            "DoorSideSidorAl-n" : Bool;   // ST2 Door sidoor Side - Output stage defective
            "DoorSideSidorAl-L" : Bool;   // ST2 Door sidoor Side - Current measurement error
            "DoorSideSidorAl-t" : Bool;   // ST2 Door sidoor Side - Belt torn
            "DoorSideSidorAl-U" : Bool;   // ST2 Door sidoor Side - Max. mass to be moved:
            "Spare 1_7" : Bool;
            CloseDoorByHand : Bool;   // ST2 Door sidoor Side - close by hand
            DoorFrontLearn : Bool;   // ST2 Doors side in learn procedure - Please Wait
            DoorSideSpecial : Bool;   // Please Wait - Sidoor Side in Special - mode The system is in an error state or special mode (system is shutting down, powering up or saving safety-related parameters)
            SidoorSideOpenAlarm : Bool;   // Sidoor Side - An obstruction was detected in the opening direction
            SidoorSideCloseAlarm : Bool;   // Sidoor Side - An obstruction was detected in the closing direction
            Temp1 : Array[4..9] of Byte;
         END_STRUCT;
         BASE : Struct   // SHUTTER
            ClampDownWP : Bool;   // ST2 Base Clamp down failed to advance I200.2/B274.8
            ClampDownPP : Bool;   // ST2 Base Clamp down failed to reverse I200.3/B274.10
            ClampDownBS : Bool;   // ST2 Base Clamp down both sensors ON I200.2-3/B274.8-10
            MobileBaseWP : Bool;   // ST2 Base Mobile base failed to advance I200.4/B274.12
            MobileBasePP : Bool;   // ST2 Base Mobile base failed to reverse I200.5/B274.14
            MobileBaseTS : Bool;   // ST2 Base Mobile base both sensors ON I200.4-5/B274.12-14
            ClampUpLeftWP : Bool;   // ST2 Base Clamp up left failed to advance I200.6/B274.16
            ClampUpLeftPP : Bool;   // ST2 Base Clamp up left failed to reverse I200.7/B274.18
            ClampUpLeftBS : Bool;   // ST2 Base Clamp up left both sensors ON I200.2-3/B274.16-18
            ClampUpRightWP : Bool;   // ST2 Base Clamp up right failed to advance I201.0/B275.4
            ClampUpRightPP : Bool;   // ST2 Base Clamp up right failed to reverse I201.1/B275.6
            ClampUpRightBS : Bool;   // ST2 Base Clamp up right both sensors ON I200.0-1/B275.4-6
            TankStopperWP : Bool;   // ST2 Tank Stopper failed to advance I231.4/B277.12
            TankStopperPP : Bool;   // ST2 Tank Stopper failed to reverse I231.5/B277.14
            TankStopperBS : Bool;   // ST2 Tank Stopper both sensors ON I231.4-5/B277.12-14
            Temp1 : Array[2..9] of Byte;
         END_STRUCT;
         ST2OP02 : Struct   // CUT FSU CONV
            UnitTransferAdvFlt : Bool;   // ST2OP02 (Cut FSU CONV) Unit Transfer Failed To Advance I220.0/B284.4
            UnitTransferRetFlt : Bool;   // ST2OP02 (Cut FSU CONV) Unit Transfer Failed To Return I220.1/B284.6
            UnitTransferTSFlt : Bool;   // ST2OP02 (Cut FSU CONV) Unit Transfer Two Sensors ON I220.0-1/B284.4-6
            CuttingAdvFlt : Bool;   // ST2OP02 (Cut FSU CONV) Cutting Cylinder Failed To Advance I220.2/B284.8
            CuttingRevFlt : Bool;   // ST2OP02 (Cut FSU CONV) Cutting Cylinder Failed To Return I220.3/B284.10
            CuttingTSFlt : Bool;   // ST2OP02 (Cut FSU CONV) Cutting Cylinder Two Sensors ON I220.2-3/B284.8-10
            ClampAdvFlt : Bool;   // ST2OP02 (Cut FSU CONV) Ring Clamp Failed To Advance I220.4/B284.12
            ClampRevFlt : Bool;   // ST2OP02 (Cut FSU CONV) Ring Clamp Failed To Return I220.5/B284.14
            ClampTSFlt : Bool;   // ST2OP02 (Cut FSU CONV) Ring Clamp Two Sensors ON I220.4-5/B284.12-14
            FingersAdvFlt : Bool;   // ST2OP02 (Cut FSU CONV) Fingers Failed To Advance I220.6/B284.16
            FingersRevFlt : Bool;   // ST2OP02 (Cut FSU CONV) Fingers Failed To Return I220.6/B284.16
            FingersTSFlt : Bool;
            Spare1_4Alm : Bool;
            Spare1_5Alm : Bool;
            Spare1_6Alm : Bool;
            Spare1_7Alm : Bool;
            SlugUnitFlt : Bool;   // ST2OP02 (Cut FSU CONV) Slug Not Detected on Unit RC300 I220.7/B284.18
            CuttingTimeOutFlt : Bool;   // ST2OP02 (Cut FSU CONV) Cutting Time Exceeded RC301
            CylFaultDuringCycleFlt : Bool;   // ST2OP02 (Cut FSU CONV) Cylinder Fault During Cycle RC302
            CycleNotFinishFlt : Bool;   // ST2OP02 (Cut FSU CONV) Cycle Failed To Finish RC303
            CycleNotStartedFlt : Bool;   // ST2OP02 (Cut FSU CONV) Cycle Not Started Fault RC304
            SlugFrameFlt : Bool;   // ST2OP02 (Cut FSU CONV) Slug Not Detected by Frame RC305 I201.3/B275.10
            CylPositionLostFlt : Bool;   // ST2OP02 (Cut FSU CONV) Cylinders Position Lost in manual RC306
            Spare2_7Alm : Bool;
            Spare3_0Alm : Bool;
            Spare3_1Alm : Bool;
            Spare3_2Alm : Bool;
            Spare3_3Alm : Bool;
            Spare3_4Alm : Bool;
            Spare3_5Alm : Bool;
            Spare3_6Alm : Bool;
            Spare3_7Alm : Bool;
            CircuitBreakerTripFlt : Bool;   // ST2OP02 (Cut FSU CONV) Circuit Breaker Tripped I26.0/F110.3
            SlugSensorOffFlt : Bool;   // ST2OP02 (Cut FSU CONV) Slug sensor OFF I220.7/B284.18
            ContactorOffFlt : Bool;   // ST2OP02 (Cut FSU CONV) Motor Contactor OFF I26.1/K145.3
            ContactorOnFlt : Bool;   // ST2OP02 (Cut FSU CONV) Motor Contactor ON I26.1/K145.3
            FrameConstantlyONFlt : Bool;   // ST2OP02 (Cut FSU CONV) Frame Constanly ON I201.3/B275.10
            ChangeKnife : Bool;   // ST2OP02 (Cut FSU CONV) Change knife
            Spare4_6Alm : Bool;
            Spare4_7Alm : Bool;
            CarStopWPAlm : Bool;   // ST2OP02 (Cut FSU CONV) Carriage stopper failed to advance I221.0/B285.4
            CarStopPPAlm : Bool;   // ST2OP02 (Cut FSU CONV) Carriage stopper failed to reverse I221.1/B285.6
            CarStopBSAlm : Bool;   // ST2OP02 (Cut FSU CONV) Carriage stopper both sensors ON I221.0-1/B285.4-6
            TrHorWPAlm : Bool;   // ST2OP02 (Cut FSU CONV) Tr horizontal failed to advance I221.2/B285.8
            TrHorPPAlm : Bool;   // ST2OP02 (Cut FSU CONV) Tr horizontal failed to reverse I221.3/B285.10
            TrHorBSAlm : Bool;   // ST2OP02 (Cut FSU CONV) Tr horizontal both sensors ON I221.2-3/B285.8-10
            Spare5_6Alm : Bool;
            SlugBoxFull : Bool;   // ST2OP02 (Cut FSU CONV) + ST2OP05 (CUT NIPPLE HV) Slug box full
            Temp1 : Array[6..9] of Byte;
         END_STRUCT;
         ST2OP03 : Struct   // NOTCHING
            TrHorAdvFlt : Bool;   // ST2OP03 (NOTCHING) Transfer Horizontal Failed To Advance I231.2/B277.8
            TrHorRetFlt : Bool;   // ST2OP03 (NOTCHING) Transfer Horizontal Failed To Return I231.3/B277.10
            TrHorTSFlt : Bool;   // ST2OP03 (NOTCHING) Transfer Horizontal Two Sensors ON I231.2-3/B277.8-10
            TrVerAdvFlt : Bool;   // ST2OP03 (NOTCHING) Transfer Vertical Failed To Advance I230.4/B276.12
            TrVerRetFlt : Bool;   // ST2OP03 (NOTCHING) Transfer Vertical Failed To Return I230.5/B276.14
            TrVerTSFlt : Bool;   // ST2OP03 (NOTCHING) Transfer Vertical Two Sensors ON I230.4-5/B276.12-14
            RotAdvFlt : Bool;   // ST2OP03 (NOTCHING) Rotation Failed To Advance I230.2/B276.8
            RotRetFlt : Bool;   // ST2OP03 (NOTCHING) Rotation Failed To Return I230.3/B276.10
            RotTSFlt : Bool;   // ST2OP03 (NOTCHING) Rotation Two Sensors ON I230.2-3/B276.8-10
            StampArmAdvFlt : Bool;   // ST2OP03 (NOTCHING) Stamp Arm Failed To Advance I231.6/B277.16
            StampArmRetFlt : Bool;   // ST2OP03 (NOTCHING) Stamp Arm Failed To Return I231.7/B277.18
            StampArmTSFlt : Bool;   // ST2OP03 (NOTCHING) Stamp Arm Two Sensors ON I231.6-8/B277.16-18
            StampAdvFlt : Bool;   // ST2OP03 (NOTCHING) Cutting Cylinder Failed To Advance I230.0/B276.4
            StampRevFlt : Bool;   // ST2OP03 (NOTCHING) Cutting Cylinder Failed To Return I230.1/B276.6
            StampTSFlt : Bool;   // ST2OP03 (NOTCHING) Cutting Cylinder Two Sensors ON I230.0-1/B276.4-6
            OperationNotCompletedCorrectlyFlt : Bool;   // ST2OP03 (NOTCHING) Operation not completed correctly RC1601
            Slug1DetectionFlt : Bool;   // ST2OP03 (NOTCHING) Slug 1 Detection on Unit Fault I230.6/B276.16 RC1600
            Slug2DetectionFlt : Bool;   // ST2OP03 (NOTCHING) Slug 2 Detection on Unit Fault I230.7/B276.18 RC1600
            Slug1StillPresent : Bool;   // ST2OP03 (NOTCHING) Slug 1 stuck in blowing system
            Slug2StillPresent : Bool;   // ST2OP03 (NOTCHING) Slug 2 stuck in blowing system
            CycleNotStarted : Bool;   // ST2OP03 (NOTCHING) Cycle Not Started
            CycleNotFinished : Bool;   // ST2OP03 (NOTCHING) Cycle Not Finished
            CycleTime : Bool;   // ST2OP03 (NOTCHING) Cycle Time too long
            Presence : Bool;   // ST2OP03 (NOTCHING) Alarm Presence
            Temp1 : Array[6..11] of Byte;
         END_STRUCT;
         ST2OP04 : Struct   // WELD / WELD FB CONV
            HeaterTransferAdvFlt : Bool;   // ST2OP04 (WELD FB CONV) Heater Transfer Failed to Advance I240.6/B293.16
            HeaterTransferRetFlt : Bool;   // ST2OP04 (WELD FB CONV) Heater Transfer Failed to Return I240.7/B293.18
            HeaterTransferTSFlt : Bool;   // ST2OP04 (WELD FB CONV) Heater Transfer Two Sensors on I240.6-7/B293.16-18
            GcylAdvHeatingFlt : Bool;   // ST2OP04 (WELD FB CONV) Gcyl Failed to Advance Heating I240.2/B293.8
            GcylAdvCoolingFlt : Bool;   // ST2OP04 (WELD FB CONV) Gcyl Failed to Advance Cooling I240.1/B293.6
            GcylAdvLoadingFlt : Bool;   // ST2OP04 (WELD FB CONV) Gcyl Failed to Advance Loading I240.0/B293.4
            GcylRetFlt : Bool;   // ST2OP04 (WELD FB CONV) Gcyl Failed to Return I240.3/B293.10
            GcylTSFlt : Bool;   // ST2OP04 (WELD FB CONV) Gcyl Two Sensors on I240.0/B293.4-I240.3/B293.10
            HcylAdvFlt : Bool;   // ST2OP04 (WELD FB CONV) Hcyl Failed to Advance I240.4/B293.12 (Ret Sensor for BC)
            HcylRevFlt : Bool;   // ST2OP04 (WELD FB CONV) Hcyl Failed to Return I240.5/B293.14
            HcylTSFlt : Bool;   // ST2OP04 (WELD FB CONV) Hcyl Two Sensors on I240.4/B293.12- I240.5/B293.14
            GripperAdvGripFlt : Bool;   // ST2OP04 (WELD FB CONV) Gripper Failed to Grip (Ungrip sensor Fault) I240.1/B257.4
            GripperRetUngripFlt : Bool;   // ST2OP04 (WELD FB CONV) Gripper Failed to Ungrip Sensor Fault I240.1/B257.4
            GripTSFlt : Bool;   // not used
            SpareCylFaultsInt0 : Int;
            SpareCylFaultsDInt0 : DInt;
            CompHeatPosFlt : Bool;   // ST2OP04 (WELD FB CONV) Component Failed To Gcyl Heating Position I240.2/B293.8 RC201/101
            TankHeatPosFlt : Bool;   // ST2OP04 (WELD FB CONV) Hotplate Failed To Hcyl Heating Position I240.4/B293.12 RC217
            CompCoolPosFlt : Bool;   // ST2OP04 (WELD FB CONV) Component Failed To Gcyl Cooling Position I240.1/B293.6 RC202/102
            OpenTimeFlt : Bool;   // ST2OP04 (WELD FB CONV) Open Time Exceeded RC203/103
            TempDuringCycleFlt : Bool;   // ST2OP04 (WELD FB CONV) Hotplate Temperature Fault During Cycle RC204/104
            ReservedRC0_5 : Bool;
            CompHeatPressFlt : Bool;   // ST2OP04 (WELD FB CONV) Component Heating Pressure Out Of Tolerance RC205/105
            ReservedRC0_7 : Bool;
            CompCoolPressFlt : Bool;   // ST2OP04 (WELD FB CONV) Component Cooling Pressure Out Of Tolerance RC206/106
            ReservedRC1_1 : Bool;
            ReservedRC1_2 : Bool;
            ReservedRC1_3 : Bool;
            ReservedRC1_4 : Bool;
            ReservedRC1_5 : Bool;
            TankHeatPressFlt : Bool;   // ST2OP04 (WELD FB CONV) Hcyl Heating Pressure Out Of Tolerance RC207/107
            ReservedRC1_7 : Bool;
            ReservedRC2_0 : Bool;
            ReservedRC2_1 : Bool;
            ReservedRC2_2 : Bool;
            ReservedRC2_3 : Bool;
            CycleNotFinishFlt : Bool;   // ST2OP04 (WELD FB CONV) Cycle Failed To Finish RC211/111
            CycleNotStartedFlt : Bool;   // ST2OP04 (WELD FB CONV) Cycle Not Started Fault RC212/112
            ReservedRC2_6 : Bool;
            ReservedRC2_7 : Bool;
            ReservedRC3_0 : Bool;
            TankHeatContactFlt : Bool;   // ST2OP04 (WELD FB CONV) Tank Heating Contact Pressure Calc Out Of Tolerance RC213/113
            ReservedRC3_2 : Bool;
            ReservedRC3_3 : Bool;
            MeltedComponentFlt : Bool;   // ST2OP04 (WELD FB CONV) Remove Melted Component From Gripper I241.2/B294.8 RC214/114
            ReservedRC3_5 : Bool;
            CylFaultDuringCycleFlt : Bool;   // ST2OP04 (WELD FB CONV) Cylinder Fault During Cycle RC215/115
            ReservedRC3_7 : Bool;
            ManualUsedFlt : Bool;   // ST2OP04 (WELD FB CONV) Manual Movements Used RC216/116
            CompPresent1AfterHeatFlt : Bool;   // ST2OP04 (WELD FB CONV) Component Present 1 Missing After Heating I241.2/B294.8 RC208/108
            CompPresent2AfterHeatFlt : Bool;   // ST2OP04 (WELD FB CONV) Component Present 2 Missing After Heating XXX RC218/118
            CompPresent3AfterHeatFlt : Bool;   // ST2OP04 (WELD FB CONV) Component Present 3 Missing After Heating Ixx.X RC219/119
            CompPresent4AfterHeatFlt : Bool;   // ST2OP04 (WELD FB CONV) Component Present 4 Missing After Heating Ixx.X RC220/240
            CompPresent5AfterHeatFlt : Bool;   // ST2OP04 (WELD FB CONV) Component Present 5 Missing After Heating Ixx.X RC221/121
            CompPresent6AfterHeatFlt : Bool;   // ST2OP04 (WELD FB CONV) Component Present 6 Missing After Heating Ixx.X RC222/122
            CompPresent7AfterHeatFlt : Bool;   // ST2OP04 (WELD FB CONV) Component Present 7 Missing After Heating Ixx.X RC223/123
            CompPresent8AfterHeatFlt : Bool;   // ST2OP04 (WELD FB CONV) Component Present 8 Missing After Heating Ixx.X RC224/124
            RemoveComponent1Flt : Bool;   // ST2OP04 (WELD FB CONV) Remove Component From Gripper (Present 1 after welding) I241.2/B294.8 RC209/109
            RemoveComponent2Flt : Bool;   // ST2OP04 (WELD FB CONV) Remove Component From Gripper (Present 2 after welding) XXX RC225/125
            RemoveComponent3Flt : Bool;   // ST2OP04 (WELD FB CONV) Remove Component From Gripper (Present 3 after welding) Ixx.X RC226/126
            RemoveComponent4Flt : Bool;   // ST2OP04 (WELD FB CONV) Remove Component From Gripper (Present 4 after welding) Ixx.X RC227/127
            RemoveComponent5Flt : Bool;   // ST2OP04 (WELD FB CONV) Remove Component From Gripper (Present 5 after welding) Ixx.X RC228/128
            RemoveComponent6Flt : Bool;   // ST2OP04 (WELD FB CONV) Remove Component From Gripper (Present 6 after welding) Ixx.X RC229/129
            RemoveComponent7Flt : Bool;   // ST2OP04 (WELD FB CONV) Remove Component From Gripper (Present 7 after welding) Ixx.X RC230/130
            RemoveComponent8Flt : Bool;   // ST2OP04 (WELD FB CONV) Remove Component From Gripper (Present 8 after welding) Ixx.X RC231/131
            CompMissing1Flt : Bool;   // ST2OP04 (WELD FB CONV) Component Present 1 Missing In Gripper I241.2/B294.8 RC210/110
            CompMissing2Flt : Bool;   // ST2OP04 (WELD FB CONV) Component Present 2 Missing In Gripper XXX RC232/132
            CompMissing3Flt : Bool;   // ST2OP04 (WELD FB CONV) Component Present 3 Missing In Gripper Ixx.X RC233/133
            CompMissing4Flt : Bool;   // ST2OP04 (WELD FB CONV) Component Present 4 Missing In Gripper Ixx.X RC234/134
            CompMissing5Flt : Bool;   // ST2OP04 (WELD FB CONV) Component Present 5 Missing In Gripper Ixx.X RC235/135
            CompMissing6Flt : Bool;   // ST2OP04 (WELD FB CONV) Component Present 6 Missing In Gripper Ixx.X RC236/136
            CompMissing7Flt : Bool;   // ST2OP04 (WELD FB CONV) Component Present 7 Missing In Gripper Ixx.X RC237/137
            CompMissing8Flt : Bool;   // ST2OP04 (WELD FB CONV) Component Present 8 Missing In Gripper Ixx.X RC238/138
            SpareFaultRC : Byte;
            HotplateTempOutFlt : Bool;   // ST2OP04 (WELD FB CONV) Hotplate Temperature Out Of Tolerance
            HotplateTempSensorFlt : Bool;   // ST2OP04 (WELD FB CONV) Hotplate Thermocouple Wire Break
            HotplateTempDiffereneceTooBigFlt : Bool;   // ST2OP04 (WELD FB CONV) Hotplate Thermocouples Difference Too Big
            Reserved0_3 : Bool;
            Reserved0_4 : Bool;
            Reserved0_5 : Bool;
            CompStuckOnTankFlt : Bool;   // ST2OP04 (WELD FB CONV) Component Stuck On Tank Must reset to Ungrip Component
            TempSetFlt : Bool;   // ST2OP04 (WELD FB CONV) Hotplate Tempearture Setpoint Out Of Range
            Reserved1_0 : Bool;
            RemoveHeatedComponentFlt : Bool;   // ST2OP04 (WELD FB CONV) Remove Heated Component
            CleanHotplatesFlt : Bool;   // ST2OP04 (WELD FB CONV) Clean Hotplates
            NoDetectionUsed : Bool;   // ST2OP04 (WELD FB CONV) No Detection Used (PLC program issue)
            SpareAlarmsDInt0 : DInt;
            HotTempChanFlt : Bool;   // ST2OP04 (WELD FB CONV) Hotplate Temperature is not changing
            Spare_1 : Bool;
            Spare_2 : Bool;
            Spare_3 : Bool;
            Spare_4 : Bool;
            Spare_5 : Bool;
            Spare_6 : Bool;
            Spare_7 : Bool;
            Spare_8 : Bool;
            Spare_9 : Bool;
            Spare_10 : Bool;
            Spare_11 : Bool;
            Spare_12 : Bool;
            Spare_13 : Bool;
            Spare_14 : Bool;
            Spare_15 : Bool;
            TrCrossdvFlt : Bool;   // ST2OP04 (WELD FB CONV) Transfer Cross failed to advance I241.4/B294.12
            TrCrossRevFlt : Bool;   // ST2OP04 (WELD FB CONV) Transfer Cross failed to reverse I241.5/B294.14
            TrCrossTsFlt : Bool;   // ST2OP04 (WELD FB CONV) Transfer Cross both sensors ON I241.4-5-2/B294.12-14
            Spare_19 : Bool;
            Spare_21 : Bool;
            Spare_20 : Bool;
            TrCrossdvFlt_1 : Bool;   // ST2OP04 (WELD FB CONV) Stopper Tr Cross failed to advance I241.6/B294.16
            TrCrossRevFlt_1 : Bool;   // ST2OP04 (WELD FB CONV) Stopper Tr Cross failed to reverse I241.7/B294.18
            TrCrossTsFlt_1 : Bool;   // ST2OP04 (WELD FB CONV) Stopper Tr Cross both sensors ON I241.6-7/B294.16-18
            Spare_25 : Bool;
            Spare_26 : Bool;
            Spare_27 : Bool;
            Spare_28 : Bool;
            Spare_29 : Bool;
            Spare_30 : Bool;
            Spare_31 : Bool;
            RemCycleNotStartedBADFromPrevStation : Bool;
            Spare_33 : Bool;
            Spare_34 : Bool;
            FailedToAutoLoad : Bool;
            Spare_36 : Bool;
            Spare_37 : Bool;
            Spare_38 : Bool;
         END_STRUCT;
         ST2OP05 : Struct   // CUT NIPPLE HV
            UnitTransferAdvFlt : Bool;   // ST2OP05 (CUT NIPPLE HV) Unit Transfer Failed To Advance I250.0/B286.4
            UnitTransferRetFlt : Bool;   // ST2OP05 (CUT NIPPLE HV) Unit Transfer Failed To Return I250.1/B286.6
            UnitTransferTSFlt : Bool;   // ST2OP05 (CUT NIPPLE HV) Unit Transfer Two Sensors ON I250.0-1/B286.4-6
            CuttingAdvFlt : Bool;   // ST2OP05 (CUT NIPPLE HV) Cutting Cylinder Failed To Advance I250.2/B286.8
            CuttingRevFlt : Bool;   // ST2OP05 (CUT NIPPLE HV) Cutting Cylinder Failed To Return I250.3/B286.10
            CuttingTSFlt : Bool;   // ST2OP05 (CUT NIPPLE HV) Cutting Cylinder Two Sensors ON I250.2-3/B286.8-10
            NeedleAdvFlt : Bool;   // ST2OP05 (CUT NIPPLE HV) Slug Needle Failed To Advance I250.4/B286.12
            NeedleRevFlt : Bool;   // ST2OP05 (CUT NIPPLE HV) Slug Needle Failed To Return I250.5/B286.14
            NeedleTSFlt : Bool;   // ST2OP05 (CUT NIPPLE HV) Slug Needle Two Sensors ON I250.4-5/B286.12-14
            SpareCylFaults : Int;
            SlugUnitFlt : Bool;   // ST2OP05 (CUT NIPPLE HV) Slug Not Detected on Unit RC350 I250.6/B286.16
            CuttingTimeOutFlt : Bool;   // ST2OP05 (CUT NIPPLE HV) Cutting Time Exceeded RC351
            CylFaultDuringCycleFlt : Bool;   // ST2OP05 (CUT NIPPLE HV) Cylinder Fault During Cycle RC352
            CycleNotFinishFlt : Bool;   // ST2OP05 (CUT NIPPLE HV) Cycle Failed To Finish RC353
            CycleNotStartedFlt : Bool;   // ST2OP05 (CUT NIPPLE HV) Cycle Not Started Fault RC354
            SlugFrameFlt : Bool;   // ST2OP05 (CUT NIPPLE HV) Slug Not Detected by Frame RC355 I201.3/B275.10
            ManualUsedFlt : Bool;   // ST2OP05 (CUT NIPPLE HV) Cylinders Position Lost in manual RC356
            Spare2_7Alm : Bool;
            Spare3_0Alm : Bool;
            BumperHorizontalWPAlm : Bool;
            BumperHorizontalPPAlm : Bool;
            BumperHorizontalBSAlm : Bool;
            Spare_8_7Alm : Bool;
            MissingStartFromSTDBlock : Bool;   // ST2OP05 (CUT NIPPLE HV) Missing Start Cycle From Standard Block
            SlugBoxFull : Bool;
            Spare3_7Alm : Bool;
            CircuitBreakerTripFlt : Bool;   // ST2OP05 (CUT NIPPLE HV) Circuit Breaker Tripped I26.2/F110.7
            SlugSensorOnFlt : Bool;   // ST2OP05 (CUT NIPPLE HV) Slug sensor ON I250.6/B286.16
            ContactorOffFlt : Bool;   // ST2OP05 (CUT NIPPLE HV) Motor Contactor OFF I26.3/K145.5
            ContactorOnFlt : Bool;   // ST2OP05 (CUT NIPPLE HV) Motor Contactor ON I26.3/K145.5
            FrameConstantlyONFlt : Bool;   // ST2OP05 (CUT NIPPLE HV) Frame Constanly ON I201.3/B275.10
            ChangeKnife : Bool;   // ST2OP05 (CUT NIPPLE HV) Change knife
            Spare4_6Alm : Bool;
            Spare4_7Alm : Bool;
            CarStopWPAlm : Bool;   // ST2OP05 (CUT NIPPLE HV) Carriage stopper failed to advance I251.0/B287.4
            CarStopPPAlm : Bool;   // ST2OP05 (CUT NIPPLE HV) Carriage stopper failed to reverse I251.1/B287.6
            CarStopBSAlm : Bool;   // ST2OP05 (CUT NIPPLE HV) Carriage stopper both sensors on I251.0-1/B287.4-6
            HorizontalTrAdvFlt : Bool;   // ST2OP05 (CUT NIPPLE HV) Transfer Horizontal failed to advance I251.2/B287.8
            HorizontalTrRetFlt : Bool;   // ST2OP05 (CUT NIPPLE HV) Transfer Horizontal failed to reverse I251.3/B287.10
            HorizontalTrTSFlt : Bool;   // ST2OP05 (CUT NIPPLE HV) Transfer Horizontal both sensors ON I251.2-3 /B287.8-10
            Spare7_6Alm : Bool;
            Spare7_7Alm : Bool;
            Spare8_0Alm : Bool;
            VacuumFlapWP : Bool;
            VacuumFlapPP : Bool;
            VacuumFlapBS : Bool;
            Spare7_6Alm_2 : Bool;
            Spare7_7Alm_2 : Bool;
            Spare8_0Alm_2 : Bool;
            Spare7_6Alm_3 : Bool;
            Spare7_7Alm_3 : Bool;
            Spare8_0Alm_3 : Bool;
            Spare7_6Alm_4 : Bool;
            Spare7_7Alm_4 : Bool;
            Spare8_0Alm_4 : Bool;
            Spare8_0Alm_5 : Bool;
            Spare8_0Alm_6 : Bool;
            Spare8_0Alm_7 : Bool;
         END_STRUCT;
         ST2OP06 : Struct   // WELD ICV HV
            HeaterTransferAdvFlt : Bool;   // ST2OP06 (WELD ICV HV) Heater Transfer Failed to Advance I260.6/B295.16
            HeaterTransferRetFlt : Bool;   // ST2OP06 (WELD ICV HV) Heater Transfer Failed to Return I260.7/B295.18
            HeaterTransferTSFlt : Bool;   // ST2OP06 (WELD ICV HV) Heater Transfer Two Sensors on I260.6-7/B295.16-18
            GcylAdvHeatingFlt : Bool;   // ST2OP06 (WELD ICV HV) Gcyl Failed to Advance Heating I260.2/B295.8
            GcylAdvCoolingFlt : Bool;   // ST2OP06 (WELD ICV HV) Gcyl Failed to Advance Cooling I260.1/B295.6
            GcylAdvLoadingFlt : Bool;   // ST2OP06 (WELD ICV HV) Gcyl Failed to Advance Loading I260.0/B295.4
            GcylRetFlt : Bool;   // ST2OP06 (WELD ICV HV) Gcyl Failed to Return I260.3/B295.10
            GcylTSFlt : Bool;   // ST2OP06 (WELD ICV HV) Gcyl Two Sensors on I260.0-3/B295.4-10
            HcylAdvFlt : Bool;   // ST2OP06 (WELD ICV HV) Hcyl Failed to Advance I260.4/B295.12
            HcylRevFlt : Bool;   // ST2OP06 (WELD ICV HV) Hcyl Failed to Return I260.5/B295.14
            HcylTSFlt : Bool;   // ST2OP06 (WELD ICV HV) Hcyl Two Sensors on I260.4-5/B295.12-14
            GripperAdvGripFlt : Bool;   // ST2OP06 (WELD ICV HV) Gripper Failed to Grip (Ungrip sensor Fault) I261.0/B296.4
            GripperRetUngripFlt : Bool;   // ST2OP06 (WELD ICV HV) Gripper Failed to Ungrip Sensor Fault I261.0/B296.4
            GripTSFlt : Bool;   // not used
            ApproachGcylAdvFlt : Bool;   // ST2OP06 (WELD ICV HV) Approach Gcyl Failed to Advance Ix.x
            ApproachGcylRetFlt : Bool;   // ST2OP06 (WELD ICV HV) Approach Gcyl Failed to Return Ix.x
            ApproachGcylTSFlt : Bool;   // ST2OP06 (WELD ICV HV) Approach Gcyl Two Sensors on Ixx.X-Ixx.X
            ApproachHcylAdvFlt : Bool;   // ST2OP06 (WELD ICV HV) Approach Hcyl Failed to Advance Ix.x
            ApproachHcylRetFlt : Bool;   // ST2OP06 (WELD ICV HV) Approach Hcyl Failed to Return Ix.x
            ApproachHcylTSFlt : Bool;   // ST2OP06 (WELD ICV HV) Approach Hcyl Two Sensors on Ixx.X-Ixx.X
            ComplGcylAdvLockFlt : Bool;   // ST2OP06 (WELD ICV HV) Compliancy Gcyl Failed to Lock Ix.x
            ComplGcylRetUnlockFlt : Bool;   // ST2OP06 (WELD ICV HV) Compliancy Gcyl Failed to Unlock Ix.x
            ComplGcylRetTSFlt : Bool;   // ST2OP06 (WELD ICV HV) Compliancy Gcyl Two Sensors on Ixx.X-Ixx.X
            ComplHcylAdvLockFlt : Bool;   // ST2OP06 (WELD ICV HV) Compliancy Hcyl Failed to Lock Ix.x
            ComplHcylRetUnlockFlt : Bool;   // ST2OP06 (WELD ICV HV) Compliancy Hcyl Failed to Unlock Ix.x
            ComplHcylRetTSFlt : Bool;   // ST2OP06 (WELD ICV HV) Compliancy Hcyl Two Sensors on Ixx.X-Ixx.X
            ComponentHeaterAdvFlt : Bool;   // ST2OP06 (WELD ICV HV) Component Heater Failed to Advance Ixx.X
            ComponentHeaterRetFlt : Bool;   // ST2OP06 (WELD ICV HV) Component Heater Failed to Return Ixx.X
            ComponentHeaterTSFlt : Bool;   // ST2OP06 (WELD ICV HV) Component Heater Two Sensors on Ixx.X-Ixx.X
            PullerAdvFlt : Bool;   // ST2OP06 (WELD ICV HV) Puller Failed to Advance Ixx.X
            PullerRetFlt : Bool;   // ST2OP06 (WELD ICV HV) Puller Failed to Return Ixx.X
            PullerTSFlt : Bool;   // ST2OP06 (WELD ICV HV) Puller Two Sensors on Ixx.X-Ixx.X
            SpareCylFaultsDInt0 : DInt;
            CompHeatPosFlt : Bool;   // ST2OP06 (WELD ICV HV) Component Failed To Gcyl Heating Position I260.2/B295.8 RC001
            TankHeatPosFlt : Bool;   // ST2OP06 (WELD ICV HV) Tank Hotplate Failed To Hcyl Heating Position I260.4/B295.12 RC002
            CompCoolPosFlt : Bool;   // ST2OP06 (WELD ICV HV) Component Failed To Gcyl Cooling Position I260.1/B295.6 RC003
            OpenTimeFlt : Bool;   // ST2OP06 (WELD ICV HV) Open Time Exceeded RC004
            TankTempDuringCycleFlt : Bool;   // ST2OP06 (WELD ICV HV) Tank Hotplate Temperature Fault During Cycle RC005
            CompMatchForwPressFlt : Bool;   // ST2OP06 (WELD ICV HV) Component Matching Forward Pressure Out Of Tolerance RC006
            CompHeatForwPressFlt : Bool;   // ST2OP06 (WELD ICV HV) Component Heating Forward Pressure Out Of Tolerance RC007
            CompJunctForwPressFlt : Bool;   // ST2OP06 (WELD ICV HV) Component Junction Forward Pressure Out Of Tolerance RC008
            CompCoolForwPressFlt : Bool;   // ST2OP06 (WELD ICV HV) Component Cooling Forward Pressure Out Of Tolerance RC009
            CompMatchBackPressFlt : Bool;   // ST2OP06 (WELD ICV HV) Component Matching Back Pressure Out Of Tolerance RC010
            CompHeatBackPressFlt : Bool;   // ST2OP06 (WELD ICV HV) Component Heat Back Pressure Out Of Tolerance RC011
            CompJunctBackPressFlt : Bool;   // ST2OP06 (WELD ICV HV) Component Junction Back Pressure Out Of Tolerance RC012
            CompCoolBackPressFlt : Bool;   // ST2OP06 (WELD ICV HV) Component Cooling Back Pressure Out Of Tolerance RC013
            TankMatchForwPressFlt : Bool;   // ST2OP06 (WELD ICV HV) Tank Matching Forward Pressure Out Of Tolerance RC014
            TankHeatForwPressFlt : Bool;   // ST2OP06 (WELD ICV HV) Tank Heating Forward Pressure Out Of Tolerance RC015
            TankMatchBackPressFlt : Bool;   // ST2OP06 (WELD ICV HV) Tank Match Back Pressure Out Of Tolerance RC016
            TankHeatBackPressFlt : Bool;   // ST2OP06 (WELD ICV HV) Tank Heat Back Pressure Out Of Tolerance RC017
            ReservedRC2_1 : Bool;
            ReservedRC2_2 : Bool;
            ReservedRC2_3 : Bool;
            CycleNotFinishFlt : Bool;   // ST2OP06 (WELD ICV HV) Cycle Failed To Finish RC021
            CycleNotStartedFlt : Bool;   // ST2OP06 (WELD ICV HV) Cycle Not Started Fault RC022
            CompMatchContactFlt : Bool;   // ST2OP06 (WELD ICV HV) Component Matching Contact Pressure Calc Out Of Tolerance RC023
            TankMatchContactFlt : Bool;   // ST2OP06 (WELD ICV HV) Tank Matching Contact Pressure Calc Out Of Tolerance RC024
            CompHeatContactFlt : Bool;   // ST2OP06 (WELD ICV HV) Component Heating Contact Pressure Calc Out Of Tolerance RC025
            TankHeatContactFlt : Bool;   // ST2OP06 (WELD ICV HV) Tank Heating Contact Pressure Calc Out Of Tolerance RC026
            CompJunctContactFlt : Bool;   // ST2OP06 (WELD ICV HV) Component Junction Contact Pressure Calc Out Of Tolerance RC027
            CompCoolContactFlt : Bool;   // ST2OP06 (WELD ICV HV) Component Cooling Contact Pressure Calc Out Of Tolerance RC028
            MeltedComponentFlt : Bool;   // ST2OP06 (WELD ICV HV) Remove Melted Component From Gripper Ix.x RC029
            CompTempDuringCycleFlt : Bool;   // ST2OP06 (WELD ICV HV) Component Hotplate Temperature Fault During Cycle RC030
            CylFaultDuringCycleFlt : Bool;   // ST2OP06 (WELD ICV HV) Cylinder Fault During Cycle RC031
            ReservedRC3_7 : Bool;
            ManualUsedFlt : Bool;   // ST2OP06 (WELD ICV HV) Manual Movements Used RC033
            LPComponentPositionChangedFlt : Bool;   // ST2OP06 (WELD ICV HV) Low Perm Component Position changed in last 5 seconds of Matching RC034
            PullerPosFlt : Bool;   // ST2OP06 (WELD ICV HV) Puller failed to Heating Position Ix.x RC035
            PullerMatchPressFlt : Bool;   // ST2OP06 (WELD ICV HV) Matching puller pressure Out of Tolerance RC036
            PullerMatchBwdPressFlt : Bool;   // ST2OP06 (WELD ICV HV) Matching puller counter pressure Out of Tolerance RC037
            PullerHeatPressFlt : Bool;   // ST2OP06 (WELD ICV HV) Heating puller pressure Out of Tolerance RC038
            PullerHeatBwdPressFlt : Bool;   // ST2OP06 (WELD ICV HV) Heating puller counter pressure Out of Tolerance RC039
            ForceOutOfTolFlagFlt : Bool;   // ST2OP06 (WELD ICV HV) Flag force out of tolerance RC040
            ForceOutOfTolBalanceFlt : Bool;   // ST2OP06 (WELD ICV HV) Balance force out of tolerance RC041
            ForceOutOfTolMatchFlt : Bool;   // ST2OP06 (WELD ICV HV) Matching force out of tolerance RC042
            ForceOutOfTolHeatFlt : Bool;   // ST2OP06 (WELD ICV HV) Heating force out of tolerance RC043
            CompPresent1AfterHeatFlt : Bool;   // ST2OP06 (WELD ICV HV) Component Present 1 Missing After Heating I261.2/B296.8 RC018
            CompPresent2AfterHeatFlt : Bool;   // ST2OP06 (WELD ICV HV) Component Present 2 Missing After Heating I261.3/B296.10 RC044
            CompPresent3AfterHeatFlt : Bool;   // ST2OP06 (WELD ICV HV) Component Present 3 Missing After Heating Ixx.X RC045
            CompPresent4AfterHeatFlt : Bool;   // ST2OP06 (WELD ICV HV) Component Present 4 Missing After Heating Ixx.X RC046
            CompPresent5AfterHeatFlt : Bool;   // ST2OP06 (WELD ICV HV) Component Present 5 Missing After Heating Ixx.X RC047
            CompPresent6AfterHeatFlt : Bool;   // ST2OP06 (WELD ICV HV) Component Present 6 Missing After Heating Ixx.X RC048
            CompPresent7AfterHeatFlt : Bool;   // ST2OP06 (WELD ICV HV) Component Present 7 Missing After Heating Ixx.X RC049
            CompPresent8AfterHeatFlt : Bool;   // ST2OP06 (WELD ICV HV) Component Present 8 Missing After Heating Ixx.X RC050
            RemoveComponent1Flt : Bool;   // ST2OP06 (WELD ICV HV) Remove Component From Gripper (Present 1 after welding) I261.2/B296.8 RC019
            RemoveComponent2Flt : Bool;   // ST2OP06 (WELD ICV HV) Remove Component From Gripper (Present 2 after welding) I261.3/B296.10 RC051
            RemoveComponent3Flt : Bool;   // ST2OP06 (WELD ICV HV) Remove Component From Gripper (Present 3 after welding) Ixx.X RC052
            RemoveComponent4Flt : Bool;   // ST2OP06 (WELD ICV HV) Remove Component From Gripper (Present 4 after welding) Ixx.X RC053
            RemoveComponent5Flt : Bool;   // ST2OP06 (WELD ICV HV) Remove Component From Gripper (Present 5 after welding) Ixx.X RC054
            RemoveComponent6Flt : Bool;   // ST2OP06 (WELD ICV HV) Remove Component From Gripper (Present 6 after welding) Ixx.X RC055
            RemoveComponent7Flt : Bool;   // ST2OP06 (WELD ICV HV) Remove Component From Gripper (Present 7 after welding) Ixx.X RC056
            RemoveComponent8Flt : Bool;   // ST2OP06 (WELD ICV HV) Remove Component From Gripper (Present 8 after welding) Ixx.X RC057
            CompMissing1Flt : Bool;   // ST2OP06 (WELD ICV HV) Component Present 1 Missing In Gripper I261.2/B296.8 RC020
            CompMissing2Flt : Bool;   // ST2OP06 (WELD ICV HV) Component Present 2 Missing In Gripper I261.3/B296.10 RC058
            CompMissing3Flt : Bool;   // ST2OP06 (WELD ICV HV) Component Present 3 Missing In Gripper Ixx.X RC059
            CompMissing4Flt : Bool;   // ST2OP06 (WELD ICV HV) Component Present 4 Missing In Gripper Ixx.X RC060
            CompMissing5Flt : Bool;   // ST2OP06 (WELD ICV HV) Component Present 5 Missing In Gripper Ixx.X RC061
            CompMissing6Flt : Bool;   // ST2OP06 (WELD ICV HV) Component Present 6 Missing In Gripper Ixx.X RC062
            CompMissing7Flt : Bool;   // ST2OP06 (WELD ICV HV) Component Present 7 Missing In Gripper Ixx.X RC063
            CompMissing8Flt : Bool;   // ST2OP06 (WELD ICV HV) Component Present 8 Missing In Gripper Ixx.X RC064
            CompPresent1Flt : Bool;   // ST2OP06 (WELD ICV HV) Component Present 1 In Gripper when Cycle Started I261.2/B296.8 RC032
            CompPresent2Flt : Bool;   // ST2OP06 (WELD ICV HV) Component Present 2 In Gripper when Cycle Started I261.3/B296.10 RC065
            CompPresent3Flt : Bool;   // ST2OP06 (WELD ICV HV) Component Present 3 In Gripper when Cycle Started Ixx.X RC066
            CompPresent4Flt : Bool;   // ST2OP06 (WELD ICV HV) Component Present 4 In Gripper when Cycle Started Ixx.X RC067
            CompPresent5Flt : Bool;   // ST2OP06 (WELD ICV HV) Component Present 5 In Gripper when Cycle Started Ixx.X RC068
            CompPresent6Flt : Bool;   // ST2OP06 (WELD ICV HV) Component Present 6 In Gripper when Cycle Started Ixx.X RC069
            CompPresent7Flt : Bool;   // ST2OP06 (WELD ICV HV) Component Present 7 In Gripper when Cycle Started Ixx.X RC070
            CompPresent8Flt : Bool;   // ST2OP06 (WELD ICV HV) Component Present 8 In Gripper when Cycle Started Ixx.X RC071
            Spare : Bool;
            Spare_1 : Bool;
            Spare_2 : Bool;
            Spare_3 : Bool;
            Spare_4 : Bool;
            CompTempOutFlt : Bool;   // ST2OP06 (WELD ICV HV) Component Hotplate Temperature Out Of Tolerance
            CompThermocoupleFlt : Bool;   // ST2OP06 (WELD ICV HV) Component Hotplate Thermocouple Wire Break
            CompTempDiffereneceTooBigFlt : Bool;   // ST2OP06 (WELD ICV HV) Component Hotplate Thermocouples Difference Too Big
            TankTempOutFlt : Bool;   // ST2OP06 (WELD ICV HV) Tank Hotplate Temperature Out Of Tolerance
            TankThermocoupleFlt : Bool;   // ST2OP06 (WELD ICV HV) Tank Hotplate Thermocouple Wire Break
            TankTempDiffereneceTooBigFlt : Bool;   // ST2OP06 (WELD ICV HV) Tank Hotplate Thermocouples Difference Too Big
            CompStuckOnTankFlt : Bool;   // ST2OP06 (WELD ICV HV) Component Stuck On Tank Must reset to Ungrip Component
            Spare_31 : Bool;
            TankTempSetFlt : Bool;   // ST2OP06 (WELD ICV HV) Tank Hotplate Temperature Setpoint Out Of Range
            RemoveHeatedComponentFlt : Bool;   // ST2OP06 (WELD ICV HV) Remove Heated Component
            CleanHotplatesFlt : Bool;   // ST2OP06 (WELD ICV HV) Clean Hotplates
            WrongConfigurationFlt : Bool;   // ST2OP06 (WELD ICV HV) Wrong option configruation of the block (PLC program issue)
            NoDetectionUsed : Bool;   // ST2OP06 (WELD ICV HV) No Detection Used (PLC program issue)
            Spare_5 : Bool;
            Spare_6 : Bool;
            CompTempSetFlt : Bool;   // ST2OP06 (WELD ICV HV) Component Hotplate Tempearture Setpoint Out Of Range
            SpareFaults : DInt;
            MobHotTempChanFlt : Bool;   // ST2OP06 (WELD ICV HV) Mobile Hotplate Temperature is not changing
            FixHotTempChanFlt : Bool;   // ST2OP06 (WELD ICV HV) Fixed Hotplate Temperature is not changing
            spare_7 : Bool;
            spare_8 : Bool;
            spare_9 : Bool;
            spare_10 : Bool;
            spare_11 : Bool;
            spare_12 : Bool;
            spare_13 : Bool;
            spare_14 : Bool;
            spare_21 : Bool;
            spare_22 : Bool;
            TrStopperVerticalWPAlm : Bool;
            TrStopperVerticalPPAlm : Bool;
            TrStopperVerticalBSAlm : Bool;
            LoadingStopperWPAlm : Bool;
            LoadingStopperPPAlm : Bool;
            LoadingStopperBSAlm : Bool;
            spare_20 : Bool;
            spare_15 : Bool;
            BadVersionComponentInGripper : Bool;
            spare_17 : Bool;
            spare_18 : Bool;
            spare_19 : Bool;
            TrCrossAdvFlt : Bool;   // ST2OP06 (WELD ICV HV) Transfer Cross failed to advance I261.4/B296.12
            TrCrossRevFlt : Bool;   // ST2OP06 (WELD ICV HV) Transfer Cross failed to reverse I261.5/B296.14
            TrCrossTsFlt : Bool;   // ST2OP06 (WELD ICV HV) Transfer Cross both sensors ON I261.4-5/B296.12-14
            spare_23 : Bool;
            StopperTrCrossAdvFlt : Bool;   // ST2OP06 (WELD ICV HV) Stopper Tr Cross failed to advance I261.6/B296.16
            StopperTrCrossRevFlt : Bool;   // ST2OP06 (WELD ICV HV) Stopper Tr Cross failed to reverse I261.7/B296.18
            StopperTrCrossTsFlt : Bool;   // ST2OP06 (WELD ICV HV) Stopper Tr Cross both sensors ON I261.6-7/B296.16-18
            spare_27 : Bool;
            RemCycleNotStartedBADFromPrevStation : Bool;
            FailedToAutoLoad : Bool;
            spare_30 : Bool;
         END_STRUCT;
         ST2OP11 : Struct   // DESTROYER
            TransferWPAlm : Bool;   // ST2OP11 (DESTROYER) Drilling transfer failed to advance I201.4/B275.12
            TransferPPAlm : Bool;   // ST2OP11 (DESTROYER) Drilling transfer failed to reverse I201.5/B275.14
            TransferBSAlm : Bool;   // ST2OP11 (DESTROYER) Drilling transfer both sensors ON I201.4-5/B275.12-14
            DrillMissing : Bool;   // ST2OP11 (DESTROYER) Drill missing I201.6/B275.16
            Spare_0_4 : Bool;
            Spare_0_5 : Bool;
            Spare_0_6 : Bool;
            Spare_0_7 : Bool;
            Spare_1_0 : Bool;
            Spare_1_1 : Bool;
            Spare_1_2 : Bool;
            Spare_1_3 : Bool;
            Spare_1_4 : Bool;
            Spare_1_5 : Bool;
            Spare_1_6 : Bool;
            Spare_1_7 : Bool;
            Temp1 : Array[2..9] of Byte;
         END_STRUCT;
         Spare : Array[20..99] of Byte;
      END_STRUCT;
      EPM : Struct
         Messages : Struct
            LoadTankA : Bool;
            LoadTankB : Bool;
            Load401component_v1 : Bool;
            Load401component_v2 : Bool;
            Load303component_v1 : Bool;
            Load303component_v2 : Bool;
            RemoveTank : Bool;
            Remove401component : Bool;
            Remove303component : Bool;
         END_STRUCT;
         Alarms : Struct
            alarm1 : Bool;
         END_STRUCT;
         Spare : Array[4..8] of Byte;
      END_STRUCT;
      zero : Int;
   END_VAR
BEGIN
END_DATA_BLOCK
